// TIA Portal project "babu_3wayTrafficLight_SIMULATION" (V15)

(* hardware
DEVICE "S7-1200 station_1"  S7-1200 Station
   slot 0: "Rack_0"  S7-1200 Rack  Rack  V1.0
   slot 1: "PLC_1"  CPU 1212C DC/DC/DC  6ES7 212-1AE40-0XB0  V4.2
*)

// ===== PLC "PLC_1"  CPU 1212C DC/DC/DC =====

VAR_GLOBAL   // PLC tag table "Default tag table"
   ""PUSH BUTTON"" AT %I0.0 : Bool;
   ""G3"" AT %Q0.0 : Bool;
   ""Y1"" AT %Q0.1 : Bool;
   ""G1"" AT %Q0.2 : Bool;
   ""R2"" AT %Q0.3 : Bool;
   ""Y2"" AT %Q0.4 : Bool;
   ""G2"" AT %Q0.5 : Bool;
   ""Y3"" AT %Q0.6 : Bool;
   ""R1"" AT %Q0.7 : Bool;
   ""R3"" AT %Q1.0 : Bool;
END_VAR